// TIA Portal V20 export
// export: Created 2026-07-10T11:12:29.221812Z, ExportSetting WithDefaults, DisplayName Totally Integrated Automation Portal, DisplayVersion V20, DisplayName TIA Portal Openness, DisplayVersion V20, DisplayName TIA Portal Version Control Interface, DisplayVersion V20, DisplayName STEP 7 Professional, DisplayVersion V20, DisplayName STEP 7 Safety, DisplayVersion V20, DisplayName WinCC Basic/Comfort/Advanced, DisplayVersion V20, DisplayName WinCC Unified, DisplayVersion V20
FUNCTION_BLOCK "ModbusClO2"   // FB26, SCL
{ S7_Optimized_Access := 'FALSE' }
VERSION : 0.1
// stored: AutoNumber true, IsIECCheckEnabled false, SetENOAutomatically false, UDAEnableTagReadback false
   VAR DB_SPECIFIC
      ProportionalDosingExternal { S7_SetPoint := 'True'} : DWord;
      AbsoluteDosing : DWord;
      SystemProductivity : DWord;
      Pressure : Word;
      Doser1Productivity : Word;
      Doser2Productivity : Word;
   END_VAR
BEGIN
   "ModbusMaster"(REQ := "ModbusLoad".DONE,
                        MB_ADDR := 1,
                        MODE := 0,
                        DATA_ADDR := 40014,
                        DATA_LEN := 1,
                        DATA_PTR := "MB".Table.ClO2.WorkMode); //OK

   "ModbusMaster"(REQ := "ModbusLoad".DONE,
         MB_ADDR := 1,
         MODE := 0,
         DATA_ADDR := 40015,
         DATA_LEN := 1,
         DATA_PTR := #Doser1Productivity);


   "MB".Table.ClO2.Doser1Productivity := #Doser1Productivity / 100;

   "ModbusMaster"(REQ := "ModbusLoad".DONE,
                 MB_ADDR := 1,
                 MODE := 0,
                 DATA_ADDR := 40016,
                 DATA_LEN := 1,
                 DATA_PTR := #Doser2Productivity);

   "MB".Table.ClO2.Doser2Productivity := #Doser2Productivity / 100;

   "ModbusMaster"(REQ := "ModbusLoad".DONE,
                 MB_ADDR := 1,
                 MODE := 0,
                 DATA_ADDR := 40020,
                 DATA_LEN := 1,
                 DATA_PTR := #Pressure);


   "MB".Table.ClO2.Pressure := #Pressure / 100;

   "ModbusMaster"(REQ := "ModbusLoad".DONE,
                 MB_ADDR := 1,
                 MODE := 0,
                 DATA_ADDR := 40025,
                 DATA_LEN := 2,
                 DATA_PTR := #SystemProductivity);

   "MB".Table.ClO2.SystemProductivity := DWORD_TO_REAL(ROL(IN := #SystemProductivity, N := 16));

   "ModbusMaster"(REQ := "ModbusLoad".DONE,
                 MB_ADDR := 1,
                 MODE := 0,
                 DATA_ADDR := 40010,
                 DATA_LEN := 1,
                 DATA_PTR := "MB".Table.ClO2.ChooseDosing); //OK

   "ModbusMaster"(REQ := "ModbusLoad".DONE,
                 MB_ADDR := 1,
                 MODE := 0,
                 DATA_ADDR := 40012,
                 DATA_LEN := 1,
                 DATA_PTR := "MB".Table.ClO2.DosersActive); //OK

   "ModbusMaster"(REQ := "ModbusLoad".DONE,
                 MB_ADDR := 1,
                 MODE := 0,
                 DATA_ADDR := 40051,
                 DATA_LEN := 2,
                 DATA_PTR := #AbsoluteDosing);

   "MB".Table.ClO2.AbsoluteDosing := DWORD_TO_REAL(ROL(IN := #AbsoluteDosing, N := 16));

   "ModbusMaster"(REQ := "ModbusLoad".DONE,
                 MB_ADDR := 1,
                 MODE := 0,
                 DATA_ADDR := 40055,
                 DATA_LEN := 2,
                 DATA_PTR := #ProportionalDosingExternal);

   "MB".Table.ClO2.ProportionalDosingExternal := DWORD_TO_REAL(ROL(IN := #ProportionalDosingExternal, N := 16));


   "ModbusMaster"(REQ := "ModbusLoad".DONE,
                 MB_ADDR := 1,
                 MODE := 0,
                 DATA_ADDR := 40011,
                 DATA_LEN := 1,
                 DATA_PTR := "MB".Table.ClO2.Alarms); //OK
END_FUNCTION_BLOCK
